{attribute 'linkalways'} 
{attribute 'no_explicit_call' := 'This FB is a CLASS and must be accessed using methods or properties'}
{attribute 'enable_dynamic_creation'}
FUNCTION_BLOCK Node_F_VN_MinElementElementwise_ULINT EXTENDS VisionNode
VAR
    ipContainer : _ITcVnContainer;
    nMin : _ULINT(0);
    hrPrev : _HRESULT(S_OK);
    hresult : _HRESULT(S_OK);
END_VAR

METHOD PUBLIC  Clone : I_Node
VAR
	pNode : POINTER TO Node_F_VN_MinElementElementwise_ULINT;
END_VAR
pNode := __NEW(Node_F_VN_MinElementElementwise_ULINT);
Clone := pNode^;
END_METHOD

METHOD FB_init : BOOL
VAR_INPUT
	bInitRetains : BOOL; // if TRUE, the retain variables are initialized (warm start / cold start)
	bInCopyCode : BOOL;  // if TRUE, the instance afterwards gets moved into the copy code (online change)
END_VAR
AddInput('ipContainer', ipContainer);
AddInput('hrPrev', hrPrev);
AddOutput('ipContainer', ipContainer);
AddOutput('nMin', nMin);
AddOutput('hresult',hresult);
END_METHOD

METHOD PROTECTED OnExecute
hresult.Value := F_VN_MinElementElementwise_ULINT(
    ipContainer := ipContainer.Value,
    nMin := nMin.Value,
    hrPrev:= hrPrev.Value);
END_METHOD

METHOD PUBLIC PreExecutionCheck
VAR_INPUT
	Check : I_PreExecutionChecks;
END_VAR
Check.IsTrue(ipContainer.IsValid, 'ipContainer must be a valid container');
Check.IsTrue(ipContainer.IsType(TC_GLOBAL_CONST_LIST.ContainerType_Vector_ULINT), 'ipContainer contains incorrect type');
END_METHOD

END_FUNCTION_BLOCK

(* stored: Version 1.1.0.1, ProductVersion 3.1.4026.13
   POU Node_F_VN_MinElementElementwise_ULINT: Id {d2fb2247-d45f-412d-bb5e-61b2bcd5b110}, SpecialFunc None
   Folder Constructor: Id {5ea28bae-f466-45d7-9096-b78da9e38830}
   Method Clone: Id {cc7ab92a-8fd3-481e-b5f0-0c18bf29c21f}
   Method FB_init: Id {2ee3c9d9-a120-4b83-bcd1-15810fa5909e}
   Method OnExecute: Id {c8715fd0-4da7-4615-8d50-cee29c9e5bfb}
   Method PreExecutionCheck: Id {4a28cbe2-89c5-4031-8465-bef13635ff31} *)
